// TIA Portal V21 export
ORGANIZATION_BLOCK "Main Richiamo Pid"   // OB35, LAD, CyclicInterrupt
TITLE = "Cyclic Interrupt"
{ S7_Optimized_Access := 'FALSE' }
// stored: AutoNumber false, SetENOAutomatically false
   VAR_TEMP
      OB35_EV_CLASS : Byte;   // Bits 0-3 = 1 (Coming event), Bits 4-7 = 1 (Event class 1)
      OB35_STRT_INF : Byte;   // 16#36 (OB 35 has started)
      OB35_PRIORITY : Byte;   // 11 (Priority of 1 is lowest)
      OB35_OB_NUMBR : Byte;   // 35 (Organization block 35, OB35)
      OB35_RESERVED_1 : Byte;   // Reserved for system
      OB35_RESERVED_2 : Byte;   // Reserved for system
      OB35_PHASE_OFFSET : Word;   // Phase offset (msec)
      OB35_RESERVED_3 : Int;   // Reserved for system
      OB35_EXC_FREQ : Int;   // Frequency of execution (msec)
      OB35_DATE_TIME : Date_And_Time;   // Date and time OB35 started
      LMN_ABS : Real;
      Appo : Real;
      FLD_ACT_ENG : Real;
      Appo_PID : Real;
      Appo_OUT : Real;
      Reset : Bool;
      PEW : Word;
      PAW : Int;
      OUT_INT : Int;
      OUT_REAL : Real;
      MinLimit : Bool;
      MaxLimit : Bool;
      "Appo Pew pid4" : Word;
      SogliaImpostataCorrettamente : Bool;
      DA_inserire : "Std_VarGestAnalog";
      VelrichiestaMotore : Int;
   END_VAR
   VAR CONSTANT
      Isteresi : Int;
   END_VAR
BEGIN

REGION Network 1 (SCL): CALL PID
   "Pid_Sterilizzatore_Pompamono"();
   "Pid_Sterilizzatore_Pompapistoni"();
   "Pid_Sterilizzatore_RaffreddamentoAcqua"();
   "Pid_Sterilizzatore_RiscaldamentoAcqua"();
   "Pid_Sterilizzatore_RiscaldamentoProdotto"();
END_REGION
END_ORGANIZATION_BLOCK
